INTERFACE ITF_Visu_Menu

METHOD PUBLIC m_SetPage : BOOL
VAR_INPUT
	i_nPage : DINT;
END_VAR
END_METHOD

PROPERTY p_nPage : DINT
GET
END_GET
END_PROPERTY

END_INTERFACE

(* stored: Version 1.1.0.1, ProductVersion 3.1.4026.13
   Itf ITF_Visu_Menu: Id {c848e96a-d8bb-4498-a5b3-d60875feeae3}
   Method m_SetPage: Id {c3829b05-6e1c-4d8c-96cd-0c36f277e77c}
   Property p_nPage: Id {2941098b-9045-4726-a412-1ffc178ed094}
   Get Get: Id {e8fb7635-c319-4f1c-be03-0eb98df6ca27} *)
